PROGRAM Main6
VAR
	Sequence:Sequence6;
	Forces:Forces6;
	Reset:Reset6;
	Faults:Faults6;
END_VAR

//Cyclic Call to the Station FBs 
Sequence();
Forces();
Reset();
Faults();

END_PROGRAM

(* stored: Version 1.1.0.1, ProductVersion 3.1.4024.11
   POU Main6: Id {cf42c77a-3f4f-4d11-8e65-60309e7f1d7b}, SpecialFunc None *)
